TEXTLIST OutputText
  0 = 'OUT00 三色灯红' | Chinese: 'OUT00 三色灯红' | English: 'OUT00 bBeacon_Red' | Vietnamese: 'OUT00 Đèn đỏ ba màu'
  1 = 'OUT01 三色灯黄' | Chinese: 'OUT01 三色灯黄' | English: 'OUT01 bBeacon_Yellow' | Vietnamese: 'OUT01 Đèn màu vàng'
  2 = 'OUT02 三色灯绿' | Chinese: 'OUT02 三色灯绿' | English: 'OUT02 bBeacon_Green' | Vietnamese: 'OUT02 Màu xanh lá cây đèn ba màu'
  3 = 'OUT03 蜂鸣器' | Chinese: 'OUT03 蜂鸣器' | English: 'OUT03 bBeacon_Buzzer' | Vietnamese: 'OUT03 buzzer'
  4 = 'OUT04 运行指示灯' | Chinese: 'OUT04 运行指示灯' | English: 'OUT04 bRuning' | Vietnamese: 'OUT04 Chạy ánh sáng'
  5 = 'OUT05 停止指示灯' | Chinese: 'OUT05 停止指示灯' | English: 'OUT05 bStop' | Vietnamese: 'OUT05 Dừng đèn'
  6 = 'OUT06 照明灯' | Chinese: 'OUT06 照明灯' | English: 'OUT06 bLED' | Vietnamese: 'OUT06 Ánh sáng'
  7 = 'OUT07 主流线分料气缸缩回' | Chinese: 'OUT07 主流线分料气缸缩回' | English: 'OUT07 bLine0Part_Cyl_H' | Vietnamese: 'OUT07 Xu hướng đường phút đoán QiGang theo lẽ'
  8 = 'OUT08 主流线分料气缸伸出' | Chinese: 'OUT08 主流线分料气缸伸出' | English: 'OUT08 bLine0Part_Cyl_W' | Vietnamese: 'OUT08 Đường phút đoán QiGang vươn ra xu hướng'
  9 = 'OUT09 主流线阻挡气缸缩回' | Chinese: 'OUT09 主流线阻挡气缸缩回' | English: 'OUT09 bLine0Prevent_Cyl_H' | Vietnamese: 'OUT09 Dòng chính ngăn chặn sự rút lại của xi lanh'
  10 = 'OUT0A 主流线阻挡气缸伸出' | Chinese: 'OUT0A 主流线阻挡气缸伸出' | English: 'OUT0A bLine0Prevent_Cyl_W' | Vietnamese: 'OUT0A Dòng chính ngăn các xi lanh thoát ra'
  11 = 'OUT0B 流水线1提升气缸缩回' | Chinese: 'OUT0B 流水线1提升气缸缩回' | English: 'OUT0B bLine1Elevator_Cyl_H' | Vietnamese: 'OUT0B 1 dây chuyền cải thiện QiGang theo lẽ'
  12 = 'OUT0C 流水线1提升气缸伸出' | Chinese: 'OUT0C 流水线1提升气缸伸出' | English: 'OUT0C bLine1Elevator_Cyl_W' | Vietnamese: 'OUT0C Xi lanh nâng ra khỏi đường ống 1'
  13 = 'OUT0D 流水线1顶升气缸缩回' | Chinese: 'OUT0D 流水线1顶升气缸缩回' | English: 'OUT0D bLine1Lift_Cyl_H' | Vietnamese: 'OUT0D Dòng 1 lít xi lanh rút lui'
  14 = 'OUT0E 流水线1顶升气缸伸出' | Chinese: 'OUT0E 流水线1顶升气缸伸出' | English: 'OUT0E bLine1Lift_Cyl_W' | Vietnamese: 'OUT0E Dây chuyền sản xuất 1 lít xi lanh thò ra'
  15 = 'OUT0F 流水线1阻挡气缸缩回' | Chinese: 'OUT0F 流水线1阻挡气缸缩回' | English: 'OUT0F bLine1Prevent_Cyl_H' | Vietnamese: 'OUT0F 1 dây chuyền ngăn cản QiGang theo lẽ'
  16 = 'OUT10 流水线1阻挡气缸伸出' | Chinese: 'OUT10 流水线1阻挡气缸伸出' | English: 'OUT10 bLine1Prevent_Cyl_W' | Vietnamese: 'OUT10 1 dây chuyền ngăn cản QiGang vươn ra'
  17 = 'OUT11 流水线1旋转气缸缩回' | Chinese: 'OUT11 流水线1旋转气缸缩回' | English: 'OUT11 bLine1Rotate_Cyl_H' | Vietnamese: 'OUT11 1 dây chuyền xoay QiGang theo lẽ'
  18 = 'OUT12 流水线1旋转气缸伸出' | Chinese: 'OUT12 流水线1旋转气缸伸出' | English: 'OUT12 bLine1Rotate_Cyl_W' | Vietnamese: 'OUT12 1 dây chuyền xoay QiGang vươn ra'
  19 = 'OUT13 流水线1调宽气缸缩回' | Chinese: 'OUT13 流水线1调宽气缸缩回' | English: 'OUT13 bLine1Adjust1_Cyl_H' | Vietnamese: 'OUT13 1 dây chuyền chuyển rộng QiGang theo lẽ'
  20 = 'OUT14 流水线1调宽气缸伸出' | Chinese: 'OUT14 流水线1调宽气缸伸出' | English: 'OUT14 bLine1Adjust1_Cyl_W' | Vietnamese: 'OUT14 1 dây chuyền chuyển rộng QiGang vươn ra'
  21 = 'OUT15 预留' | Chinese: 'OUT15 预留' | English: 'OUT15 None1' | Vietnamese: 'OUT15 Dành riêng'
  22 = 'OUT16 预留' | Chinese: 'OUT16 预留' | English: 'OUT16 None2' | Vietnamese: 'OUT16 Dành riêng'
  23 = 'OUT17 流水线2顶升气缸缩回' | Chinese: 'OUT17 流水线2顶升气缸缩回' | English: 'OUT17 bLine2Lift_Cyl_H' | Vietnamese: 'OUT17 2 dây chuyền trên đỉnh lít QiGang theo lẽ'
  24 = 'OUT18 流水线2顶升气缸伸出' | Chinese: 'OUT18 流水线2顶升气缸伸出' | English: 'OUT18 bLine2Lift_Cyl_W' | Vietnamese: 'OUT18 Dây chuyền 2 lít QiGang vươn ra'
  25 = 'OUT19 流水线2阻挡气缸缩回' | Chinese: 'OUT19 流水线2阻挡气缸缩回' | English: 'OUT19 bLine2Prevent_Cyl_H' | Vietnamese: 'OUT19 Dây chuyền 2 ngăn cản QiGang theo lẽ'
  26 = 'OUT1A 流水线2阻挡气缸伸出' | Chinese: 'OUT1A 流水线2阻挡气缸伸出' | English: 'OUT1A bLine2Prevent_Cyl_W' | Vietnamese: 'OUT1A Dây chuyền 2 ngăn cản QiGang vươn ra'
  27 = 'OUT1B 流水线2校平气缸1缩回' | Chinese: 'OUT1B 流水线2校平气缸1缩回' | English: 'OUT1B bLine2Standard1_Cyl_H' | Vietnamese: 'OUT1B 1 dây chuyền 2 trường phẳng QiGang theo lẽ'
  28 = 'OUT1C 流水线2校平气缸1伸出' | Chinese: 'OUT1C 流水线2校平气缸1伸出' | English: 'OUT1C bLine2Standard1_Cyl_W' | Vietnamese: 'OUT1C 1 dây chuyền 2 trường phẳng QiGang vươn ra'
  29 = 'OUT1D 流水线2校平气缸2缩回' | Chinese: 'OUT1D 流水线2校平气缸2缩回' | English: 'OUT1D bLine2Standard2_Cyl_H' | Vietnamese: 'OUT1D Dây chuyền 2 trường QiGang giới phẳng 2 theo lẽ'
  30 = 'OUT1E 流水线2校平气缸2伸出' | Chinese: 'OUT1E 流水线2校平气缸2伸出' | English: 'OUT1E bLine2Standard2_Cyl_W' | Vietnamese: 'OUT1E 2 trường QiGang giới phẳng 2 dây chuyền vươn ra'
  31 = 'OUT1F 流水线2解锁侧推气缸1缩回' | Chinese: 'OUT1F 流水线2解锁侧推气缸1缩回' | English: 'OUT1F bLine2OpenLateral1_Cyl_H' | Vietnamese: 'OUT1F Dây chuyền 2 bỏ khóa đẩy QiGang 1 theo lẽ bên hông'
  32 = 'OUT20 流水线2解锁侧推气缸1伸出' | Chinese: 'OUT20 流水线2解锁侧推气缸1伸出' | English: 'OUT20 bLine2OpenLateral1_Cyl_W' | Vietnamese: 'OUT20 Dây chuyền 2 bỏ khóa đẩy QiGang 1 bên hông vươn ra'
  33 = 'OUT21 流水线2解锁旋转气缸缩回' | Chinese: 'OUT21 流水线2解锁旋转气缸缩回' | English: 'OUT21 bLine2OpenRotate_Cyl_H' | Vietnamese: 'OUT21 Dây chuyền 2 mở khóa xoay QiGang theo lẽ'
  34 = 'OUT22 流水线2解锁旋转气缸伸出' | Chinese: 'OUT22 流水线2解锁旋转气缸伸出' | English: 'OUT22 bLine2OpenRotate_Cyl_W' | Vietnamese: 'OUT22 Dây chuyền 2 mở khóa xoay QiGang vươn ra'
  35 = 'OUT23 流水线2解锁侧推气缸2缩回' | Chinese: 'OUT23 流水线2解锁侧推气缸2缩回' | English: 'OUT23 bLine2OpenLateral2_Cyl_H' | Vietnamese: 'OUT23 Dây chuyền 2 bỏ khóa đẩy QiGang bên hông 2 theo lẽ'
  36 = 'OUT24 流水线2解锁侧推气缸2伸出' | Chinese: 'OUT24 流水线2解锁侧推气缸2伸出' | English: 'OUT24 bLine2OpenLateral2_Cyl_W' | Vietnamese: 'OUT24 Dây chuyền 2 bỏ khóa đẩy QiGang 2 bên hông vươn ra'
  37 = 'OUT25 预留' | Chinese: 'OUT25 预留' | English: 'OUT25 None202' | Vietnamese: 'OUT25 Dành riêng'
  38 = 'OUT26 预留' | Chinese: 'OUT26 预留' | English: 'OUT26 None203' | Vietnamese: 'OUT26 Dành riêng'
  39 = 'OUT27 流水线3上料位顶升缩回' | Chinese: 'OUT27 流水线3上料位顶升缩回' | English: 'OUT27 bLine3LoadLift_Cyl_H' | Vietnamese: 'OUT27 Dây chuyền đoán người trên 3 lít theo lẽ'
  40 = 'OUT28 流水线3上料位顶升伸出' | Chinese: 'OUT28 流水线3上料位顶升伸出' | English: 'OUT28 bLine3LoadLift_Cyl_W' | Vietnamese: 'OUT28 Dây chuyền đoán người trên 3 lít vươn ra'
  41 = 'OUT29 流水线3上料位阻挡缩回' | Chinese: 'OUT29 流水线3上料位阻挡缩回' | English: 'OUT29 bLine3LoadPrevent_Cyl_H' | Vietnamese: 'OUT29 Dây chuyền trên 3 đoán ngăn cản theo lẽ'
  42 = 'OUT2A 流水线3上料位阻挡伸出' | Chinese: 'OUT2A 流水线3上料位阻挡伸出' | English: 'OUT2A bLine3LoadPrevent_Cyl_W' | Vietnamese: 'OUT2A Dây chuyền trên 3 đoán ai ngăn cản'
  43 = 'OUT2B 流水线3上料位旋转缩回' | Chinese: 'OUT2B 流水线3上料位旋转缩回' | English: 'OUT2B bLine3LoadRotate_Cyl_H' | Vietnamese: 'OUT2B Dây chuyền trên 3 đoán xoay theo lẽ'
  44 = 'OUT2C 流水线3上料位旋转伸出' | Chinese: 'OUT2C 流水线3上料位旋转伸出' | English: 'OUT2C bLine3LoadRotate_Cyl_W' | Vietnamese: 'OUT2C Dây chuyền trên 3 đoán xoay vươn ra'
  45 = 'OUT2D 流水线3解锁位顶升缩回' | Chinese: 'OUT2D 流水线3解锁位顶升缩回' | English: 'OUT2D bLine3OpenLift_Cyl_H' | Vietnamese: 'OUT2D 3 đội bỏ khóa một cái dây chuyền lít theo lẽ'
  46 = 'OUT2E 流水线3解锁位顶升伸出' | Chinese: 'OUT2E 流水线3解锁位顶升伸出' | English: 'OUT2E bLine3OpenLift_Cyl_W' | Vietnamese: 'OUT2E Dây chuyền, mở khóa 3 đội một cái lít vươn ra'
  47 = 'OUT2F 流水线3解锁位阻挡缩回' | Chinese: 'OUT2F 流水线3解锁位阻挡缩回' | English: 'OUT2F bLine3OpenPrevent_Cyl_H' | Vietnamese: 'OUT2F Dây chuyền, mở khóa 3 người ngăn cản theo lẽ'
  48 = 'OUT30 流水线3解锁位阻挡伸出' | Chinese: 'OUT30 流水线3解锁位阻挡伸出' | English: 'OUT30 bLine3OpenPrevent_Cyl_W' | Vietnamese: 'OUT30 Dây chuyền, mở khóa 3 người ngăn cản ngươi ra'
  49 = 'OUT31 流水线3校平气缸1缩回' | Chinese: 'OUT31 流水线3校平气缸1缩回' | English: 'OUT31 bLine3Standard1_Cyl_H' | Vietnamese: 'OUT31 3 trường QiGang giới phẳng dây chuyền 1 theo lẽ'
  50 = 'OUT32 流水线3校平气缸1伸出' | Chinese: 'OUT32 流水线3校平气缸1伸出' | English: 'OUT32 bLine3Standard1_Cyl_W' | Vietnamese: 'OUT32 1 dây chuyền 3 trường phẳng QiGang vươn ra'
  51 = 'OUT33 流水线3校平气缸2缩回' | Chinese: 'OUT33 流水线3校平气缸2缩回' | English: 'OUT33 bLine3Standard2_Cyl_H' | Vietnamese: 'OUT33 3 trường QiGang giới phẳng dây chuyền 2 theo lẽ'
  52 = 'OUT34 流水线3校平气缸2伸出' | Chinese: 'OUT34 流水线3校平气缸2伸出' | English: 'OUT34 bLine3Standard2_Cyl_W' | Vietnamese: 'OUT34 3 trường QiGang giới phẳng dây chuyền 2 vươn ra'
  53 = 'OUT35 流水线3解锁侧推气缸1缩回' | Chinese: 'OUT35 流水线3解锁侧推气缸1缩回' | English: 'OUT35 bLine3OpenLateral1_Cyl_H' | Vietnamese: 'OUT35 Dây chuyền, mở khóa 3 đẩy QiGang 1 theo lẽ bên hông'
  54 = 'OUT36 流水线3解锁侧推气缸1伸出' | Chinese: 'OUT36 流水线3解锁侧推气缸1伸出' | English: 'OUT36 bLine3OpenLateral1_Cyl_W' | Vietnamese: 'OUT36 Dây chuyền, mở khóa 3 đẩy QiGang 1 bên hông vươn ra'
  55 = 'OUT37 流水线3解锁旋转气缸缩回' | Chinese: 'OUT37 流水线3解锁旋转气缸缩回' | English: 'OUT37 bLine3OpenRotate_Cyl_H' | Vietnamese: 'OUT37 Dây chuyền, mở khóa 3 xoay QiGang theo lẽ'
  56 = 'OUT38 流水线3解锁旋转气缸伸出' | Chinese: 'OUT38 流水线3解锁旋转气缸伸出' | English: 'OUT38 bLine3OpenRotate_Cyl_W' | Vietnamese: 'OUT38 Dây chuyền, mở khóa 3 xoay QiGang vươn ra'
  57 = 'OUT39 流水线3解锁侧推气缸2缩回' | Chinese: 'OUT39 流水线3解锁侧推气缸2缩回' | English: 'OUT39 bLine3OpenLateral2_Cyl_H' | Vietnamese: 'OUT39 3 dây chuyền 2 theo lẽ bỏ khóa đẩy QiGang bên hông'
  58 = 'OUT3A 流水线3解锁侧推气缸2伸出' | Chinese: 'OUT3A 流水线3解锁侧推气缸2伸出' | English: 'OUT3A bLine3OpenLateral2_Cyl_W' | Vietnamese: 'OUT3A Dây chuyền, mở khóa 3 đẩy QiGang 2 bên hông vươn ra'
  59 = 'OUT3B 预留' | Chinese: 'OUT3B 预留' | English: 'OUT3B None200' | Vietnamese: 'OUT3B Dành riêng'
  60 = 'OUT3C 预留' | Chinese: 'OUT3C 预留' | English: 'OUT3C None201' | Vietnamese: 'OUT3C Dành riêng'
  61 = 'OUT3D 取料模组升降气缸1缩回' | Chinese: 'OUT3D 取料模组升降气缸1缩回' | English: 'OUT3D bTakeLift1_Cyl_H' | Vietnamese: 'OUT3D Lấy đoán trông QiGang phản lực lên nhóm 1 theo lẽ'
  62 = 'OUT3E 取料模组升降气缸1伸出' | Chinese: 'OUT3E 取料模组升降气缸1伸出' | English: 'OUT3E bTakeLift1_Cyl_W' | Vietnamese: 'OUT3E Lấy khối nâng xi lanh 1 thò ra'
  63 = 'OUT3F 取料模组升降气缸2缩回' | Chinese: 'OUT3F 取料模组升降气缸2缩回' | English: 'OUT3F bTakeLift2_Cyl_H' | Vietnamese: 'OUT3F Lấy đoán trông QiGang phản lực lên nhóm 2 theo lẽ'
  64 = 'OUT40 取料模组升降气缸2伸出' | Chinese: 'OUT40 取料模组升降气缸2伸出' | English: 'OUT40 bTakeLift2_Cyl_W' | Vietnamese: 'OUT40 Lấy đoán trông QiGang phản lực lên nhóm 2'
  65 = 'OUT41 取料模组夹紧气缸缩回' | Chinese: 'OUT41 取料模组夹紧气缸缩回' | English: 'OUT41 bTakeClamp_Cyl_H' | Vietnamese: 'OUT41 Lấy mô-đun kẹp xi lanh rút lui'
  66 = 'OUT42 取料模组夹紧气缸伸出' | Chinese: 'OUT42 取料模组夹紧气缸伸出' | English: 'OUT42 bTakeClamp_Cyl_W' | Vietnamese: 'OUT42 Lấy đoán trông kẹp chặt QiGang vươn ra nhóm'
  67 = 'OUT43 下UC模组升降气缸缩回' | Chinese: 'OUT43 下UC模组升降气缸缩回' | English: 'OUT43 bUcLift_Cyl_H' | Vietnamese: 'OUT43 Tiếp theo và trông QiGang phản lực lên nhóm theo lẽ'
  68 = 'OUT44 下UC模组升降气缸伸出' | Chinese: 'OUT44 下UC模组升降气缸伸出' | English: 'OUT44 bUcLift_Cyl_W' | Vietnamese: 'OUT44 Xi lanh nâng theo mô-đun UC thò ra'
  69 = 'OUT45 下UC模组夹紧气缸缩回' | Chinese: 'OUT45 下UC模组夹紧气缸缩回' | English: 'OUT45 bUcClamp_Cyl_H' | Vietnamese: 'OUT45 Nhóm tiếp theo và trông kẹp chặt QiGang theo lẽ'
  70 = 'OUT46 下UC模组夹紧气缸伸出' | Chinese: 'OUT46 下UC模组夹紧气缸伸出' | English: 'OUT46 bUcClamp_Cyl_W' | Vietnamese: 'OUT46 Các xi lanh bị kẹp dưới mô-đun UC thò ra'
  71 = 'OUT47 下UC模组摆动气缸缩回' | Chinese: 'OUT47 下UC模组摆动气缸缩回' | English: 'OUT47 bUcSwing_Cyl_H' | Vietnamese: 'OUT47 Mô-đun UC dưới đang quay xi lanh'
  72 = 'OUT48 下UC模组摆动气缸伸出' | Chinese: 'OUT48 下UC模组摆动气缸伸出' | English: 'OUT48 bUcSwing_Cyl_W' | Vietnamese: 'OUT48 Các xi lanh xoay trong mô-đun UC phía dưới thò ra'
  73 = 'OUT49 下UC升降气缸1缩回' | Chinese: 'OUT49 下UC升降气缸1缩回' | English: 'OUT49 bUcLift1_Cyl_H' | Vietnamese: 'OUT49 Xi lanh nâng dưới UC 1 rút lui'
  74 = 'OUT4A 下UC升降气缸1伸出' | Chinese: 'OUT4A 下UC升降气缸1伸出' | English: 'OUT4A bUcLift1_Cyl_W' | Vietnamese: 'OUT4A Xi lanh nâng dưới UC 1 thò ra'
  75 = 'OUT4B 下UC夹紧气缸1缩回' | Chinese: 'OUT4B 下UC夹紧气缸1缩回' | English: 'OUT4B bUcClamp1_Cyl_H' | Vietnamese: 'OUT4B Khóa xi lanh 1 lại'
  76 = 'OUT4C 下UC夹紧气缸1伸出' | Chinese: 'OUT4C 下UC夹紧气缸1伸出' | English: 'OUT4C bUcClamp1_Cyl_W' | Vietnamese: 'OUT4C Bên dưới ống 1 được mở ra'
  77 = 'OUT4D 下UC旋转气缸1缩回' | Chinese: 'OUT4D 下UC旋转气缸1缩回' | English: 'OUT4D bUcRotate1_Cyl_H' | Vietnamese: 'OUT4D Xi lanh quay dưới UC 1 rút lui'
  78 = 'OUT4E 下UC旋转气缸1伸出' | Chinese: 'OUT4E 下UC旋转气缸1伸出' | English: 'OUT4E bUcRotate1_Cyl_W' | Vietnamese: 'OUT4E Xi lanh quay dưới UC 1 thò ra'
  79 = 'OUT4F 下UC升降气缸2缩回' | Chinese: 'OUT4F 下UC升降气缸2缩回' | English: 'OUT4F bUcLift2_Cyl_H' | Vietnamese: 'OUT4F Xi lanh nâng 2 co lại'
  80 = 'OUT50 下UC升降气缸2伸出' | Chinese: 'OUT50 下UC升降气缸2伸出' | English: 'OUT50 bUcLift2_Cyl_W' | Vietnamese: 'OUT50 QiGang phản lực lên xuống và giơ 2'
  81 = 'OUT51 下UC夹紧气缸2缩回' | Chinese: 'OUT51 下UC夹紧气缸2缩回' | English: 'OUT51 bUcClamp2_Cyl_H' | Vietnamese: 'OUT51 Quay lại xi lanh 2'
  82 = 'OUT52 下UC夹紧气缸2伸出' | Chinese: 'OUT52 下UC夹紧气缸2伸出' | English: 'OUT52 bUcClamp2_Cyl_W' | Vietnamese: 'OUT52 Bên dưới ống 2 được mở ra'
  83 = 'OUT53 下UC旋转气缸2缩回' | Chinese: 'OUT53 下UC旋转气缸2缩回' | English: 'OUT53 bUcRotate2_Cyl_H' | Vietnamese: 'OUT53 Xi lanh quay dưới UC 2 rút lại'
  84 = 'OUT54 下UC旋转气缸2伸出' | Chinese: 'OUT54 下UC旋转气缸2伸出' | English: 'OUT54 bUcRotate2_Cyl_W' | Vietnamese: 'OUT54 Xi lanh 2 quay dưới UC thò ra'
  85 = 'OUT55 下UC皮带推料气缸缩回' | Chinese: 'OUT55 下UC皮带推料气缸缩回' | English: 'OUT55 bUcDrive_Cyl_H' | Vietnamese: 'OUT55 Co lại xi lanh đẩy dưới vành đai UC'
  86 = 'OUT56 下UC皮带推料气缸伸出' | Chinese: 'OUT56 下UC皮带推料气缸伸出' | English: 'OUT56 bUcDrive_Cyl_W' | Vietnamese: 'OUT56 Các xi lanh đẩy ra ngoài'
  87 = 'OUT57 下工装提升气缸1缩回' | Chinese: 'OUT57 下工装提升气缸1缩回' | English: 'OUT57 bFrockElevator1_Cyl_H' | Vietnamese: 'OUT57 Máy nâng xi lanh 1 rút lui'
  88 = 'OUT58 下工装提升气缸1伸出' | Chinese: 'OUT58 下工装提升气缸1伸出' | English: 'OUT58 bFrockElevator1_Cyl_W' | Vietnamese: 'OUT58 Nâng cao GongZhuang tiếp theo là 1 QiGang vươn ra'
  89 = 'OUT59 下工装旋转压紧气缸1缩回' | Chinese: 'OUT59 下工装旋转压紧气缸1缩回' | English: 'OUT59 bFrockRotateDown1_Cyl_H' | Vietnamese: 'OUT59 Tải trọng xoay xi lanh 1 co lại'
  90 = 'OUT5A 下工装旋转压紧气缸1伸出' | Chinese: 'OUT5A 下工装旋转压紧气缸1伸出' | English: 'OUT5A bFrockRotateDown1_Cyl_W' | Vietnamese: 'OUT5A Công cụ xoay xi lanh 1 căng ra'
  91 = 'OUT5B 下工装拨料气缸1缩回' | Chinese: 'OUT5B 下工装拨料气缸1缩回' | English: 'OUT5B bFrockPush1_Cyl_H' | Vietnamese: 'OUT5B Xi lanh số 1 thu hồi'
  92 = 'OUT5C 下工装拨料气缸1伸出' | Chinese: 'OUT5C 下工装拨料气缸1伸出' | English: 'OUT5C bFrockPush1_Cyl_W' | Vietnamese: 'OUT5C Xi lanh máy đo 1 thò ra'
  93 = 'OUT5D 下工装提升气缸2缩回' | Chinese: 'OUT5D 下工装提升气缸2缩回' | English: 'OUT5D bFrockElevator2_Cyl_H' | Vietnamese: 'OUT5D Máy nâng xi lanh 2 rút lui'
  94 = 'OUT5E 下工装提升气缸2伸出' | Chinese: 'OUT5E 下工装提升气缸2伸出' | English: 'OUT5E bFrockElevator2_Cyl_W' | Vietnamese: 'OUT5E Máy nâng xi lanh 2 thò ra'
  95 = 'OUT5F 下工装旋转压紧气缸2缩回' | Chinese: 'OUT5F 下工装旋转压紧气缸2缩回' | English: 'OUT5F bFrockRotateDown2_Cyl_H' | Vietnamese: 'OUT5F Công cụ xoay xi lanh 2 nén lại'
  96 = 'OUT60 下工装旋转压紧气缸2伸出' | Chinese: 'OUT60 下工装旋转压紧气缸2伸出' | English: 'OUT60 bFrockRotateDown2_Cyl_W' | Vietnamese: 'OUT60 Công cụ xoay xi lanh 2 căng ra'
  97 = 'OUT61 下工装拨料气缸2缩回' | Chinese: 'OUT61 下工装拨料气缸2缩回' | English: 'OUT61 bFrockPush2_Cyl_H' | Vietnamese: 'OUT61 Xi lanh theo tải trọng 2 rút lui'
  98 = 'OUT62 下工装拨料气缸2伸出' | Chinese: 'OUT62 下工装拨料气缸2伸出' | English: 'OUT62 bFrockPush2_Cyl_W' | Vietnamese: 'OUT62 Xi lanh máy đo 2 thò ra'
  99 = 'OUT63 下工装皮带推料气缸缩回' | Chinese: 'OUT63 下工装皮带推料气缸缩回' | English: 'OUT63 bFrockBelt_Cyl_H' | Vietnamese: 'OUT63 Tải trọng vành đai đẩy xi lanh rút lui'
  100 = 'OUT64 下工装皮带推料气缸伸出' | Chinese: 'OUT64 下工装皮带推料气缸伸出' | English: 'OUT64 bFrockBelt_Cyl_W' | Vietnamese: 'OUT64 Tải vành đai đẩy ra khỏi xi lanh'
  101 = 'OUT65 预留' | Chinese: 'OUT65 预留' | English: 'OUT65 None3' | Vietnamese: 'OUT65 Dành riêng'
  102 = 'OUT66 流水线1皮带运行' | Chinese: 'OUT66 流水线1皮带运行' | English: 'OUT66 bLine1Axis' | Vietnamese: 'OUT66 Dây chuyền sản xuất 1 chạy'
  103 = 'OUT67 流水线2皮带运行' | Chinese: 'OUT67 流水线2皮带运行' | English: 'OUT67 bLine2Axis' | Vietnamese: 'OUT67 Dây chuyền sản xuất 2 chạy'
  104 = 'OUT68 流水线3皮带运行' | Chinese: 'OUT68 流水线3皮带运行' | English: 'OUT68 bLine3Axis' | Vietnamese: 'OUT68 Dây chuyền sản xuất 3 vành đai chạy'
  105 = 'OUT69 下UC皮带运行' | Chinese: 'OUT69 下UC皮带运行' | English: 'OUT69 bUnloadUCLine' | Vietnamese: 'OUT69 Cảnh sát chìm đang chạy'
  106 = 'OUT6A 下工装皮带运行' | Chinese: 'OUT6A 下工装皮带运行' | English: 'OUT6A bUnloadElevatorLine' | Vietnamese: 'OUT6A Vành đai công cụ chạy'
  107 = 'OUT6B 预留' | Chinese: 'OUT6B 预留' | English: 'OUT6B None9' | Vietnamese: 'OUT6B Dành riêng'
  108 = 'OUT6C 预留' | Chinese: 'OUT6C 预留' | English: 'OUT6C None10' | Vietnamese: 'OUT6C Dành riêng'
  109 = 'OUT6D 预留' | Chinese: 'OUT6D 预留' | English: 'OUT6D None11' | Vietnamese: 'OUT6D Dành riêng'
  110 = 'OUT6E 预留' | Chinese: 'OUT6E 预留' | English: 'OUT6E None12' | Vietnamese: 'OUT6E Dành riêng'
  111 = 'OUT6F 预留' | Chinese: 'OUT6F 预留' | English: 'OUT6F None13' | Vietnamese: 'OUT6F Dành riêng'
   = ''
END_TEXTLIST

(* stored: Version 1.1.0.1, ProductVersion 3.1.4024.3
   TextList OutputText: Id {3e72ff28-dbe1-48a8-be85-75c7936f53c1} *)
